KUKA KRL program: test.src, test.dat

--- test.src ---
&ACCESS RVO
DEF TEST()
;FOLD INI
  ;FOLD BASISTECH INI
    GLOBAL INTERRUPT DECL 3 WHEN $STOPMESS==TRUE DO IR_STOPM ( )
    INTERRUPT ON 3
    BAS (#INITMOV,0 )
  ;ENDFOLD (BASISTECH INI)
  ;FOLD USER INI
  ;Make your modifications here

  ;ENDFOLD (USER INI)
;ENDFOLD (INI)

; Generated by AUTODESK Fusion 360 CAM 2.0.14793
; Creation date: Thursday, March 16, 2023 18:51:23

; Set PTP velocity and acceleration
$VEL_AXIS[1] = 25
$VEL_AXIS[2] = 25
$VEL_AXIS[3] = 25
$VEL_AXIS[4] = 25
$VEL_AXIS[5] = 25
$VEL_AXIS[6] = 25
$ACC_AXIS[1] = 20
$ACC_AXIS[2] = 20
$ACC_AXIS[3] = 20
$ACC_AXIS[4] = 20
$ACC_AXIS[5] = 20
$ACC_AXIS[6] = 20

; To set 'Tool On Robot' Mode
$IPO_MODE = #BASE

; Set smoothing value
$APO.CDIS = 2

; Set $ADVANCE value (number of points read in advance)
$ADVANCE = 3

; Set BASE
$BASE = BASE_DATA[1]

; Spindle OFF
;SPINDLE_OFF()

END

--- test.dat ---
&ACCESS RVO
DEFDAT test
;FOLD EXTERNAL DECLARATIONS;%{PE}%MKUKATPBASIS,%CEXT,%VCOMMON,%P
  ;FOLD BASISTECH EXT;%{PE}%MKUKATPBASIS,%CEXT,%VEXT,%P
    EXT  BAS (BAS_COMMAND  :IN,REAL  :IN )
  ;ENDFOLD (BASISTECH EXT)

  EXT sPlanen2()
  EXT sTasche1()
  EXT sParallel2()
  EXT sKontur5()

;ENDFOLD (EXTERNAL DECLARATIONS)
ENDDAT
